FUNCTION F_ArrayInt : ARRAY [1..NO_OF_INT_PARAM] OF INT
VAR_INPUT
	iParam		: ARRAY [1..NO_OF_INT_PARAM] OF INT;
	iParam1		: INT;
	//sParam		: ARRAY [1..NO_OF_STRING_PARAM] OF STRING;
	//bParam		: ARRAY [1..NO_OF_BOOL_PARAM] OF BOOL;
	//dParam		: ARRAY [1..NO_OF_LREAL_PARAM] OF LREAL;
END_VAR

	F_ArrayInt := iParam;
	F_ArrayInt[1] := iParam1;

END_FUNCTION

(* stored: Version 1.1.0.1, ProductVersion 3.1.4022.18
   POU F_ArrayInt: Id {05662d80-7966-4112-b307-ed766fb9b3b2}, SpecialFunc None *)
